FUNCTION_BLOCK FB_W_STRING (* Converts a WSTRING to its STRING equivalent *)
  (* Standard: 61499-1; Classification: Strings; Function: Conversion; Type: WSTRING to STRING *)
  (* Version 0.0, 2007-08-17, JHC, Holobloc Inc *)
  (* Compiler header: package fb.rt.strings; *)
  (* Compiler classdef: SimpleFB *)
  (* Compiler Java Sun JDK 1.6.0 *)
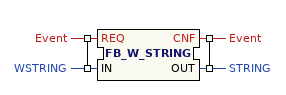
  EVENT_INPUT
    REQ WITH IN; (* Normal Execution Request *)
  END_EVENT
  EVENT_OUTPUT
    CNF WITH OUT; (* Execution Confirmation *)
  END_EVENT
  VAR_INPUT
    IN : WSTRING;
  END_VAR
  VAR_OUTPUT
    OUT : STRING;
  END_VAR
  ALGORITHM REQ IN Java:
OUT.value = IN.value.getBytes();
OUT.length = OUT.value.length;
  END_ALGORITHM
END_FUNCTION_BLOCK
